Fanuc KAREL source: kb00032.KL

-- PROVISIONAL review KL for V940-1; original PC SHA256 1f6ae709d04269e05f369fd7c7e60765b0b4e9d1b1b3f6ab8f795d76632a03af
-- Incomplete behavior may be omitted. Consult companion uncertainty JSON. Do not deploy.
PROGRAM KB00032
%NOLOCKGROUP
BEGIN
  -- V9_ZERO_TABLE_METADATA_HINT layout=0002_ascii; no indexed target words; source/name/runtime held
  -- UNRESOLVED_PC offsets 5-14; opcodes 3F,75
  -- UNRESOLVED_PC offsets 19-28; opcodes 3F,75
  -- UNRESOLVED_PC offsets 33-40; opcodes 9D,23
  -- UNRESOLVED_PC offsets 45-71; opcodes 27,22,2A,22,2A,22,31
  -- UNRESOLVED_PC offsets 76-80; opcodes 7F
END KB00032
